# EPICS substitutions: TRITON/TRITON-IOC-01App/Db/TRITON_pressure_channels.substitutions
file TRITON_temp_channels.template {

pattern {PORT, P, CHAN}
{"\$(PORT)", "\$(P)", "P1"}
{"\$(PORT)", "\$(P)", "P2"}
{"\$(PORT)", "\$(P)", "P3"}
{"\$(PORT)", "\$(P)", "P5"}
}
